(* IEC 61131-3 sources: volt/packages/volt-lsp-iec/test-corpus/bakon-nano/Device/Plc Logic/Application/Library Manager/CmpIoMgr Implementation, 47 files *)

(* ---- IOMGRCONFIGGETCONNECTOR.pou ---- *)
FUNCTION IOMGRCONFIGGETCONNECTOR : POINTER TO IoConfigConnector
VAR_INPUT
	PCONNECTORLIST : POINTER TO IoConfigConnector;
	PNCOUNT : POINTER TO DINT;
	DWMODULETYPE : DWORD;
	DWINSTANCE : DWORD;
END_VAR
END_FUNCTION

(* ---- IOMGRCONFIGGETCONNECTORBYDRIVER.pou ---- *)
FUNCTION IOMGRCONFIGGETCONNECTORBYDRIVER : POINTER TO IoConfigConnector
VAR_INPUT
	PIBASE : IBase;
	BIECDRIVER : DINT;
	NINDEX : DINT;
	PRESULT : POINTER TO RTS_IEC_RESULT;
END_VAR
END_FUNCTION

(* ---- IOMGRCONFIGGETCONNECTORLIST.pou ---- *)
FUNCTION IOMGRCONFIGGETCONNECTORLIST : RTS_IEC_RESULT
VAR_INPUT
	PPCONNECTORLIST : POINTER TO POINTER TO IoConfigConnector;
	PNCOUNT : POINTER TO DINT;
END_VAR
END_FUNCTION

(* ---- IOMGRCONFIGGETDRIVER.pou ---- *)
FUNCTION IOMGRCONFIGGETDRIVER : IBase
VAR_INPUT
	PCONNECTOR : POINTER TO IoConfigConnector;
	PBIECDRIVER : POINTER TO DINT;
	PRESULT : POINTER TO RTS_IEC_RESULT;
END_VAR
END_FUNCTION

(* ---- IOMGRCONFIGGETFIRSTCHILD.pou ---- *)
FUNCTION IOMGRCONFIGGETFIRSTCHILD : POINTER TO IoConfigConnector
VAR_INPUT
	PCONNECTORLIST : POINTER TO IoConfigConnector;
	PNCOUNT : POINTER TO DINT;
	PFATHER : POINTER TO IoConfigConnector;
END_VAR
END_FUNCTION

(* ---- IOMGRCONFIGGETFIRSTCONNECTOR.pou ---- *)
FUNCTION IOMGRCONFIGGETFIRSTCONNECTOR : POINTER TO IoConfigConnector
VAR_INPUT
	PCONNECTORLIST : POINTER TO IoConfigConnector;
	PNCOUNT : POINTER TO DINT;
	WTYPE : WORD;
END_VAR
END_FUNCTION

(* ---- IOMGRCONFIGGETNEXTCHILD.pou ---- *)
FUNCTION IOMGRCONFIGGETNEXTCHILD : POINTER TO IoConfigConnector
VAR_INPUT
	PCONNECTORLIST : POINTER TO IoConfigConnector;
	PNCOUNT : POINTER TO DINT;
	PFATHER : POINTER TO IoConfigConnector;
END_VAR
END_FUNCTION

(* ---- IOMGRCONFIGGETNEXTCONNECTOR.pou ---- *)
FUNCTION IOMGRCONFIGGETNEXTCONNECTOR : POINTER TO IoConfigConnector
VAR_INPUT
	PCONNECTORLIST : POINTER TO IoConfigConnector;
	PNCOUNT : POINTER TO DINT;
	WTYPE : WORD;
END_VAR
END_FUNCTION

(* ---- IOMGRCONFIGGETPARAMETER.pou ---- *)
FUNCTION IOMGRCONFIGGETPARAMETER : POINTER TO IoConfigParameter
VAR_INPUT
	PCONNECTOR : POINTER TO IoConfigConnector;
	DWPARAMETERID : DWORD;
END_VAR
END_FUNCTION

(* ---- IOMGRCONFIGGETPARAMETERVALUEBYTE.pou ---- *)
FUNCTION IOMGRCONFIGGETPARAMETERVALUEBYTE : BYTE
VAR_INPUT
	PPARAMETER : POINTER TO IoConfigParameter;
	PRESULT : POINTER TO UDINT;
END_VAR
END_FUNCTION

(* ---- IOMGRCONFIGGETPARAMETERVALUEDWORD.pou ---- *)
FUNCTION IOMGRCONFIGGETPARAMETERVALUEDWORD : DWORD
VAR_INPUT
	PPARAMETER : POINTER TO IoConfigParameter;
	PRESULT : POINTER TO UDINT;
END_VAR
END_FUNCTION

(* ---- IOMGRCONFIGGETPARAMETERVALUEPOINTER.pou ---- *)
FUNCTION IOMGRCONFIGGETPARAMETERVALUEPOINTER : POINTER TO BYTE
VAR_INPUT
	PPARAMETER : POINTER TO IoConfigParameter;
	PRESULT : POINTER TO UDINT;
END_VAR
END_FUNCTION

(* ---- IOMGRCONFIGGETPARAMETERVALUEWORD.pou ---- *)
FUNCTION IOMGRCONFIGGETPARAMETERVALUEWORD : WORD
VAR_INPUT
	PPARAMETER : POINTER TO IoConfigParameter;
	PRESULT : POINTER TO UDINT;
END_VAR
END_FUNCTION

(* ---- IOMGRCONFIGRESETDIAGNOSIS.pou ---- *)
FUNCTION IOMGRCONFIGRESETDIAGNOSIS : UDINT
VAR_INPUT
	PCONNECTOR : POINTER TO IoConfigConnector;
	DWFLAGS : DWORD;
END_VAR
END_FUNCTION

(* ---- IOMGRCONFIGSETDIAGNOSIS.pou ---- *)
FUNCTION IOMGRCONFIGSETDIAGNOSIS : UDINT
VAR_INPUT
	PCONNECTOR : POINTER TO IoConfigConnector;
	DWFLAGS : DWORD;
END_VAR
END_FUNCTION

(* ---- IOMGRCOPYINPUTBE.pou ---- *)
FUNCTION IOMGRCOPYINPUTBE : RTS_IEC_RESULT
VAR_INPUT
	PCHANNEL : POINTER TO IoConfigChannelMap;
	PADDRESS : POINTER TO BYTE;
END_VAR
END_FUNCTION

(* ---- IOMGRCOPYINPUTLE.pou ---- *)
FUNCTION IOMGRCOPYINPUTLE : RTS_IEC_RESULT
VAR_INPUT
	PCHANNEL : POINTER TO IoConfigChannelMap;
	PADDRESS : POINTER TO BYTE;
END_VAR
END_FUNCTION

(* ---- IOMGRCOPYOUTPUTBE.pou ---- *)
FUNCTION IOMGRCOPYOUTPUTBE : RTS_IEC_RESULT
VAR_INPUT
	PCHANNEL : POINTER TO IoConfigChannelMap;
	PADDRESS : POINTER TO BYTE;
END_VAR
END_FUNCTION

(* ---- IOMGRCOPYOUTPUTLE.pou ---- *)
FUNCTION IOMGRCOPYOUTPUTLE : RTS_IEC_RESULT
VAR_INPUT
	PCHANNEL : POINTER TO IoConfigChannelMap;
	PADDRESS : POINTER TO BYTE;
END_VAR
END_FUNCTION

(* ---- IOMGRGETBUSCYCLETYPE.pou ---- *)
FUNCTION IOMGRGETBUSCYCLETYPE : UDINT
VAR_INPUT
	PCONNECTOR : POINTER TO IoConfigConnector;
	PRESULT : POINTER TO RTS_IEC_RESULT;
END_VAR
END_FUNCTION

(* ---- IOMGRGETCONFIGAPPLICATION.pou ---- *)
FUNCTION IOMGRGETCONFIGAPPLICATION : RTS_IEC_RESULT
VAR_INPUT
	PSZCONFIGAPPLICATION : REFERENCE TO STRING;
	PNMAXLEN : POINTER TO DINT;
END_VAR
END_FUNCTION

(* ---- IOMGRGETDRIVERPROPERTIES.pou ---- *)
FUNCTION IOMGRGETDRIVERPROPERTIES : RTS_IEC_RESULT
VAR_INPUT
	HIODRV : RTS_IEC_HANDLE;
	PPPROPERTIES : POINTER TO POINTER TO DWORD;
END_VAR
END_FUNCTION

(* ---- IOMGRGETFIRSTDRIVERINSTANCE.pou ---- *)
FUNCTION IOMGRGETFIRSTDRIVERINSTANCE : IBase
VAR_INPUT
	PBIECDRIVER : POINTER TO DINT;
	PRESULT : POINTER TO RTS_IEC_RESULT;
END_VAR
END_FUNCTION

(* ---- IOMGRGETMODULEDIAGNOSIS.pou ---- *)
FUNCTION IOMGRGETMODULEDIAGNOSIS : UDINT
VAR_INPUT
	PCONNECTOR : POINTER TO IoConfigConnector;
END_VAR
END_FUNCTION

(* ---- IOMGRGETNEXTDRIVERINSTANCE.pou ---- *)
FUNCTION IOMGRGETNEXTDRIVERINSTANCE : IBase
VAR_INPUT
	PIBASEPREV : IBase;
	PBIECDRIVER : POINTER TO DINT;
	PRESULT : POINTER TO RTS_IEC_RESULT;
END_VAR
END_FUNCTION

(* ---- IOMGRIDENTIFY.pou ---- *)
FUNCTION IOMGRIDENTIFY : UDINT
VAR_INPUT
	PCONNECTOR : POINTER TO IoConfigConnector;
END_VAR
END_FUNCTION

(* ---- IOMGRLOCKENTER.pou ---- *)
FUNCTION IOMGRLOCKENTER : RTS_IEC_RESULT
VAR_INPUT
	HIODRV : RTS_IEC_HANDLE;
	DWLOCKSCOPE : DWORD;
END_VAR
END_FUNCTION

(* ---- IOMGRLOCKLEAVE.pou ---- *)
FUNCTION IOMGRLOCKLEAVE : RTS_IEC_RESULT
VAR_INPUT
	HIODRV : RTS_IEC_HANDLE;
	DWLOCKSCOPE : DWORD;
END_VAR
END_FUNCTION

(* ---- IOMGRREADINPUTS.pou ---- *)
FUNCTION IOMGRREADINPUTS : UDINT
VAR_INPUT
	PTASKMAP : POINTER TO IoConfigTaskMap;
END_VAR
END_FUNCTION

(* ---- IOMGRREADPARAMETER.pou ---- *)
FUNCTION IOMGRREADPARAMETER : UDINT
VAR_INPUT
	DWMODULETYPE : DWORD;
	DWINSTANCE : DWORD;
	DWPARAMETERID : DWORD;
	PDATA : POINTER TO BYTE;
	DWBITSIZE : DWORD;
	DWBITOFFSET : DWORD;
END_VAR
END_FUNCTION

(* ---- IOMGRRECONFIGURE.pou ---- *)
FUNCTION IOMGRRECONFIGURE : RTS_IEC_RESULT
VAR_INPUT
	PCONNECTOR : POINTER TO IoConfigConnector;
	PUDISTATE : POINTER TO UDINT;
END_VAR
END_FUNCTION

(* ---- IOMGRREGISTERCONFIGAPPLICATION.pou ---- *)
FUNCTION IOMGRREGISTERCONFIGAPPLICATION : RTS_IEC_RESULT
VAR_INPUT
	PSZCONFIGAPPLICATION : REFERENCE TO STRING;
END_VAR
END_FUNCTION

(* ---- IOMGRREGISTERINSTANCE2.pou ---- *)
FUNCTION IOMGRREGISTERINSTANCE2 : RTS_IEC_HANDLE
VAR_INPUT
	DWCLASSID : DWORD;
	PITF : IBase;
	PRESULT : POINTER TO RTS_IEC_RESULT;
END_VAR
END_FUNCTION

(* ---- IOMGRSCANMODULES.pou ---- *)
FUNCTION IOMGRSCANMODULES : UDINT
VAR_INPUT
	PCONNECTOR : POINTER TO IoConfigConnector;
	PPCONNECTORLIST : POINTER TO POINTER TO IoConfigConnector;
	PNCOUNT : POINTER TO DINT;
END_VAR
END_FUNCTION

(* ---- IOMGRSETDRIVERPROPERTIES.pou ---- *)
FUNCTION IOMGRSETDRIVERPROPERTIES : RTS_IEC_RESULT
VAR_INPUT
	HIODRV : RTS_IEC_HANDLE;
	ULPROPERTIES : DWORD;
END_VAR
END_FUNCTION

(* ---- IOMGRSETDRIVERPROPERTY.pou ---- *)
FUNCTION IOMGRSETDRIVERPROPERTY : RTS_IEC_RESULT
VAR_INPUT
	HIODRV : RTS_IEC_HANDLE;
	ULPROPERTY : DWORD;
	BVALUE : DINT;
END_VAR
END_FUNCTION

(* ---- IOMGRSTARTBUSCYCLE.pou ---- *)
FUNCTION IOMGRSTARTBUSCYCLE : UDINT
VAR_INPUT
	PCONNECTOR : POINTER TO IoConfigConnector;
END_VAR
END_FUNCTION

(* ---- IOMGRSTARTBUSCYCLE2.pou ---- *)
FUNCTION IOMGRSTARTBUSCYCLE2 : UDINT
VAR_INPUT
	PCONNECTOR : POINTER TO IoConfigConnector;
	DWTYPE : UDINT;
END_VAR
END_FUNCTION

(* ---- IOMGRUNREGISTERCONFIGAPPLICATION.pou ---- *)
FUNCTION IOMGRUNREGISTERCONFIGAPPLICATION : RTS_IEC_RESULT
VAR_INPUT
	PSZCONFIGAPPLICATION : REFERENCE TO STRING;
END_VAR
END_FUNCTION

(* ---- IOMGRUNREGISTERINSTANCE.pou ---- *)
FUNCTION IOMGRUNREGISTERINSTANCE : RTS_IEC_RESULT
VAR_INPUT
	HINTERFACE : RTS_IEC_HANDLE;
END_VAR
END_FUNCTION

(* ---- IOMGRUPDATECONFIGURATION.pou ---- *)
FUNCTION IOMGRUPDATECONFIGURATION : UDINT
VAR_INPUT
	PCONNECTORLIST : POINTER TO IoConfigConnector;
	NCOUNT : DINT;
END_VAR
END_FUNCTION

(* ---- IOMGRUPDATECONFIGURATION2.pou ---- *)
FUNCTION IOMGRUPDATECONFIGURATION2 : UDINT
VAR_INPUT
	PCONNECTORLIST : POINTER TO IoConfigConnector;
	NCOUNT : DINT;
	PSZCONFIGAPPLICATION : REFERENCE TO STRING;
END_VAR
END_FUNCTION

(* ---- IOMGRUPDATEMAPPING.pou ---- *)
FUNCTION IOMGRUPDATEMAPPING : UDINT
VAR_INPUT
	PTASKMAPLIST : POINTER TO IoConfigTaskMap;
	NCOUNT : DINT;
END_VAR
END_FUNCTION

(* ---- IOMGRUPDATEMAPPING2.pou ---- *)
FUNCTION IOMGRUPDATEMAPPING2 : UDINT
VAR_INPUT
	PTASKMAPLIST : POINTER TO IoConfigTaskMap;
	NCOUNT : DINT;
	PSZCONFIGAPPLICATION : REFERENCE TO STRING;
END_VAR
END_FUNCTION

(* ---- IOMGRWATCHDOGTRIGGER.pou ---- *)
FUNCTION IOMGRWATCHDOGTRIGGER : UDINT
VAR_INPUT
	PCONNECTOR : POINTER TO IoConfigConnector;
END_VAR
END_FUNCTION

(* ---- IOMGRWRITEOUTPUTS.pou ---- *)
FUNCTION IOMGRWRITEOUTPUTS : UDINT
VAR_INPUT
	PTASKMAP : POINTER TO IoConfigTaskMap;
END_VAR
END_FUNCTION

(* ---- IOMGRWRITEPARAMETER.pou ---- *)
FUNCTION IOMGRWRITEPARAMETER : UDINT
VAR_INPUT
	DWMODULETYPE : DWORD;
	DWINSTANCE : DWORD;
	DWPARAMETERID : DWORD;
	PDATA : POINTER TO BYTE;
	DWBITSIZE : DWORD;
	DWBITOFFSET : DWORD;
END_VAR
END_FUNCTION
